(* PLC project OOP_Curso, Beckhoff Automation GmbH TwinCAT PLC Control 3.5.13.21 *)
(* stored: creationDateTime 2023-04-30T12:55:15.3953781, modificationDateTime 2023-04-30T12:55:15.4031851 *)

INTERFACE I_Calculate
METHOD Clear : I_Calculate
END_METHOD
METHOD DecreaseBy : I_Calculate
VAR_INPUT
	lDecreaseBy : REAL;
END_VAR
END_METHOD
METHOD DivideBy : I_Calculate
VAR_INPUT
	lDivideBy : REAL;
END_VAR
END_METHOD
METHOD GetResult : LREAL
VAR_INPUT
END_VAR
END_METHOD
METHOD IncreaseBy : I_Calculate
VAR_INPUT
	lIncreaseBy : REAL;
END_VAR
END_METHOD
METHOD MultiplyBy : I_Calculate
VAR_INPUT
	lMultiplyBy : REAL;
END_VAR
END_METHOD
METHOD SetNumber : I_Calculate
VAR_INPUT
	lNumber : LREAL;
END_VAR
END_METHOD
END_INTERFACE

INTERFACE I_Clear
METHOD Clear : I_SetNumber
END_METHOD
END_INTERFACE

INTERFACE I_Operation EXTENDS I_SetNumber
METHOD DecreaseBy : I_Operation
VAR_INPUT
	lDecreaseBy : REAL;
END_VAR
END_METHOD
METHOD DivideBy : I_Operation
VAR_INPUT
	lDivideBy : REAL;
END_VAR
END_METHOD
METHOD GetResult : LREAL
END_METHOD
METHOD IncreaseBy : I_Operation
VAR_INPUT
	lIncreaseBy : REAL;
END_VAR
END_METHOD
METHOD MultiplyBy : I_Operation
VAR_INPUT
	lMultiplyBy : REAL;
END_VAR
END_METHOD
END_INTERFACE

INTERFACE I_SetNumber
METHOD SetNumber : I_Operation
VAR_INPUT
	lNumber : LREAL;
END_VAR
END_METHOD
END_INTERFACE

FUNCTION_BLOCK FB_Calculate IMPLEMENTS I_Calculate
VAR
	{attribute  'hide'}
	lResult : LREAL := 0;
END_VAR

            
          

METHOD Clear : I_Calculate
                  MEMSET(destAddr:= ADR(lResult),fillByte :=0, n:=SIZEOF(lResult));
Clear := THIS^;
                
END_METHOD

METHOD DecreaseBy : I_Calculate
VAR_INPUT
	lDecreaseBy : REAL;
END_VAR
                  lResult := lResult - lDecreaseBy;
DecreaseBy := THIS^;
                
END_METHOD

METHOD DivideBy : I_Calculate
VAR_INPUT
	lDivideBy : REAL;
END_VAR
                  IF lDivideBy = 0 THEN
	lResult := 0;
ELSE	
	lResult := lResult / lDivideBy;
END_IF

DivideBy := THIS^;
                
END_METHOD

METHOD GetResult : LREAL
                  GetResult := lResult;
                
END_METHOD

METHOD IncreaseBy : I_Calculate
VAR_INPUT
	lIncreaseBy : REAL;
END_VAR
                  lResult := lResult + lIncreaseBy;
IncreaseBy := THIS^;
                
END_METHOD

METHOD MultiplyBy : I_Calculate
VAR_INPUT
	lMultiplyBy : REAL;
END_VAR
                  lResult := lResult * lMultiplyBy;
MultiplyBy := THIS^;
                
END_METHOD

METHOD SetNumber : I_Calculate
VAR_INPUT
	lNumber : LREAL;
END_VAR
                  lResult := lNumber;
SetNumber := THIS^;
                
END_METHOD
END_FUNCTION_BLOCK

FUNCTION_BLOCK FB_Calcul IMPLEMENTS I_Clear, I_SetNumber, I_Operation

VAR
	{attribute  'hide'}
	lResult : LREAL := 0;
END_VAR

            
          

METHOD Clear : I_SetNumber
                  MEMSET(destAddr:= ADR(lResult),fillByte :=0, n:=SIZEOF(lResult));
Clear := THIS^;
                
END_METHOD

METHOD SetNumber : I_Operation
VAR_INPUT
	lNumber	: LREAL;
END_VAR
                  lResult := lNumber;
SetNumber := THIS^;
                
END_METHOD

METHOD GetResult : LREAL
                  GetResult := lResult;
                
END_METHOD

METHOD DecreaseBy : I_Operation
VAR_INPUT
	lDecreaseBy	: REAL;
END_VAR
                  lResult := lResult - lDecreaseBy;
DecreaseBy := THIS^;
                
END_METHOD

{warning 'Agregar implementación de método'}
METHOD DivideBy : I_Operation
VAR_INPUT
	lDivideBy	: REAL;
END_VAR
                  IF lDivideBy = 0 THEN
	lResult := 0;
ELSE	
	lResult := lResult / lDivideBy;
END_IF

DivideBy := THIS^;
                
END_METHOD

METHOD IncreaseBy : I_Operation
VAR_INPUT
	lIncreaseBy	: REAL;
END_VAR
                  lResult := lResult + lIncreaseBy;
IncreaseBy := THIS^;
                
END_METHOD

METHOD MultiplyBy : I_Operation
VAR_INPUT
	lMultiplyBy	: REAL;
END_VAR
                  lResult := lResult * lMultiplyBy;
MultiplyBy := THIS^;
                
END_METHOD
END_FUNCTION_BLOCK

PROGRAM _14_Interface_Fluida
VAR
	fMyResult1 : LREAL;
	fbCalculate : FB_Calculate;
	
	fMyResult2 : LREAL;
	fbCalcul : FB_Calcul;
END_VAR

            // 14_1 : se ha realizado un ejemplo de interface fluida.
fMyResult1 := fbCalculate.Clear()
		            		.SetNumber(12)
		        			.DecreaseBy(2)
		        			.IncreaseBy(3.9)
	                		.MultiplyBy(5)
		        			.DivideBy(3)
		        			.GetResult();
						
// 14_2 : se ha optimazado un poco, para que la interfaz fluida no deje ir encadenando metodos que se contradigan entre si...	
// por ejemplo el metodo SetNumber() solo tiene sentido después del metodo Clear()..
// y los metodos de realizar operaciones solo tienen sentido si ha realizado antes el metodo SetNumber()...					
fMyResult2 := fbCalcul.Clear()
						.SetNumber(12)
						.DecreaseBy(2)
		        		.IncreaseBy(3.9)
	                	.MultiplyBy(5)
		        		.DivideBy(3)						
						.GetResult();

// 14_3 : la forma mas optima sería que primero de todo solo pidiese el metodo Clear() y despues solo saliese el metodo SetNumber() y después ya se pudiesen poner solo los metodos de operaciones y el de GetResult()

					
          
END_PROGRAM
